KUKA KRL data list: kuros.dat

&ACCESS RVP
&REL 159
&PARAM TEMPLATE = C:\KRC\Roboter\Template\vorgabe
&PARAM EDITMASK = *
DEFDAT  KUROS
INT mh_response_stream_ms=20
INT mh_robot_status=4
INT mh_in_traject_id=6
INT mh_out_traject_id=0
INT mh_frame_type=1
ENDDAT
